PROGRAM Process
VAR
	ProcessBlock_Tram: ProcessBlock;
	ButRight:BOOL;
	ButLeft:BOOL;
END_VAR

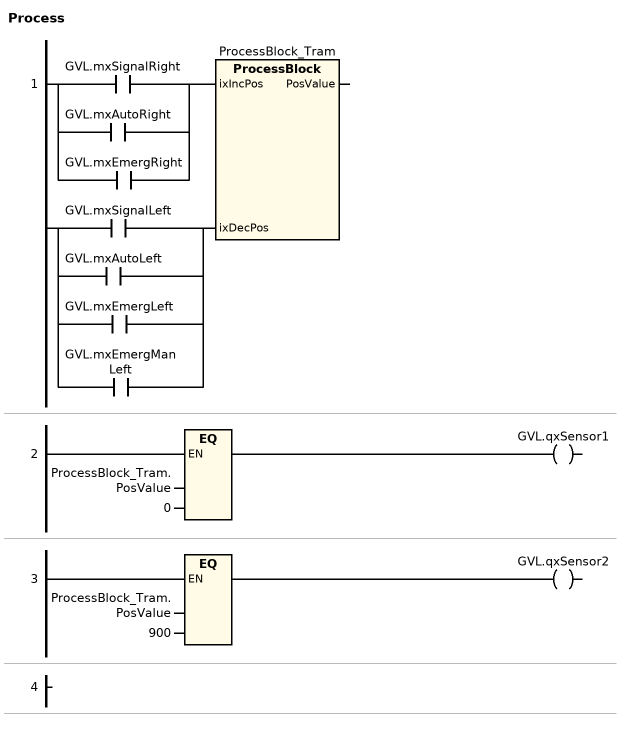
// NETWORK 1
ProcessBlock_Tram(ixIncPos := GVL.mxSignalRight OR GVL.mxAutoRight OR GVL.mxEmergRight, ixDecPos := GVL.mxSignalLeft OR GVL.mxAutoLeft OR GVL.mxEmergLeft OR GVL.mxEmergManLeft); // ProcessBlock

// NETWORK 2
GVL.qxSensor1 := ProcessBlock_Tram.PosValue = 0;

// NETWORK 3
GVL.qxSensor2 := ProcessBlock_Tram.PosValue = 900;

// NETWORK 4

END_PROGRAM

(* stored: Version 1.1.0.1, ProductVersion 3.1.4024.12
   POU Process: Id {27cd51b8-14a4-4e67-b4d4-eb08198bbcb8}, SpecialFunc None *)
